// TIA Portal V20 export
TYPE "typeVisionRetryHmiInterface"
// stored: Access Published, Namespace Unit1.Em9
   STRUCT
      currentCount : Int;
      processCount : Int := 0;
   END_STRUCT;
END_TYPE
